Staubli VAL3: iCryoShortIn.pgx

public program iCryoShortIn(num& nNum[] (dimensions=1))
begin
  nNum=dioGet(iCryoShortIn)
end
